// TIA Portal V21 export
VAR_GLOBAL   // PLC tag table "KAllComunicazione"
END_VAR
VAR_GLOBAL CONSTANT   // user constants
   KAllComun_PUT_Alarm : Int := 1;   // PUT_Alarm
   KAllComun_Get_Alarm : Int := 2;   // Get_Alarm
   KAllComun_Watchdog : Int := 5;   // Watchdog
END_VAR
